// TwinCAT 3 PLC project Prg_Arrays
// ProgramVersion: 3.1.4023.0
// libraries:
//   Tc2_Standard, * (Beckhoff Automation GmbH)
//   Tc2_System, * (Beckhoff Automation GmbH)
//   Tc3_Module, * (Beckhoff Automation GmbH)
// project tree:
//   / PlcTask.TcTTO
//   POUs/ MAIN.TcPOU, Prog_Arrays.TcPOU
// real-time tasks:
//   TASK PlcTask: cycle T#10ms, priority 20, ADS port 350

CONFIGURATION Prg_Arrays
    RESOURCE PLC ON TwinCAT3
        TASK PlcTask(INTERVAL := T#10ms, PRIORITY := 20);
        PROGRAM MAIN WITH PlcTask : MAIN;
    END_RESOURCE
END_CONFIGURATION

// ---- POUs/MAIN.TcPOU
PROGRAM MAIN
VAR
END_VAR

Prog_Arrays();

END_PROGRAM

// ---- POUs/Prog_Arrays.TcPOU
PROGRAM Prog_Arrays
VAR
	Buttons: ARRAY[1..4] OF BOOL := [4(TRUE)];
	AnalogSensor: ARRAY [1..4] OF INT := [8, 6, 7, 5];
	Coils: ARRAY [1..4] OF BOOL;
END_VAR

IF Buttons[1] = TRUE AND AnalogSensor[1] > 6 THEN
	Coils[1]:=TRUE;
END_IF

IF Buttons[2] = TRUE AND AnalogSensor[2] > 6 THEN
	Coils[2]:=TRUE;
END_IF

IF Buttons[3] = TRUE AND AnalogSensor[3] > 6 THEN
	Coils[3]:=TRUE;
END_IF

IF Buttons[4] = TRUE AND AnalogSensor[4] > 6 THEN
	Coils[4]:=TRUE;
END_IF

END_PROGRAM
